% RSLogix 500 project Arithmetic Operations.RSS, saved by version 8.30.00.16 %
PROJECT "UNTITLED"    % processor: Bul.1763 MicroLogix 1100 Series B %

PROGRAM FILES
  LAD 2   3 rungs

DATA FILES
  O0 OUTPUT  4 elements
  I1 INPUT  6 elements
  S2 STATUS  66 elements
  B3 BINARY  1 elements
  T4 TIMER  1 elements
  C5 COUNTER  1 elements
  R6 CONTROL  1 elements
  N7 INTEGER  6 elements
  F8 FLOAT  1 elements

LADDER 2
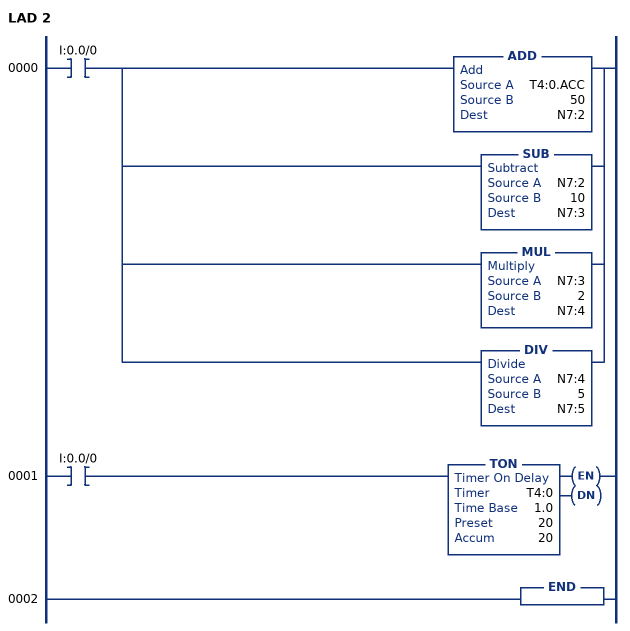
% Rung: 0 %
SOR XIC I:0.0/0 BST ADD T4:0.ACC 50 N7:2 NXB SUB N7:2 10 N7:3 NXB MUL N7:3 2 N7:4 NXB DIV N7:4 5 N7:5 BND EOR
% Rung: 1 %
SOR XIC I:0.0/0 TON T4:0 1.0 20 20 EOR
% Rung: 2 %
SOR END EOR

DATA TABLE (non-zero values as saved)
DATA T4
% .PRE .ACC %
% T4:0 % 20 20
DATA N7
% N7:0 % 10 60 70 60 120 24
